PROGRAM SoftIO
VAR
END_VAR

(*S_FEE_KMONO_PIP_01.xOn := S_FEE_KMONO_PIP_01_xON;
S_FEE_PIP_02.xOn := S_FEE_PIP_02_xON ;
S_FEE_M1L_PIP_01.xOn := S_FEE_M1L_PIP_01_xON;
S_FEE_PIP_03.xOn := S_FEE_PIP_03_xON;*)

END_PROGRAM

(* stored: Version 1.1.0.1, ProductVersion 3.1.4020.12
   POU SoftIO: Id {f0450cc5-4a7b-4096-8753-bb01176cde07}, SpecialFunc None *)
